TYPE DUT_Command :
STRUCT
	CommandType: DUT_CommandType;
	CommandString: STRING(GVL.COMMAND_LEN);
	CommandComment: STRING;
END_STRUCT
END_TYPE

(* stored: Version 1.1.0.1
   DUT DUT_Command: Id {bc90f47c-5d1d-4a76-b85b-4fab785a8038} *)
